ABB RAPID module: Module1.mod

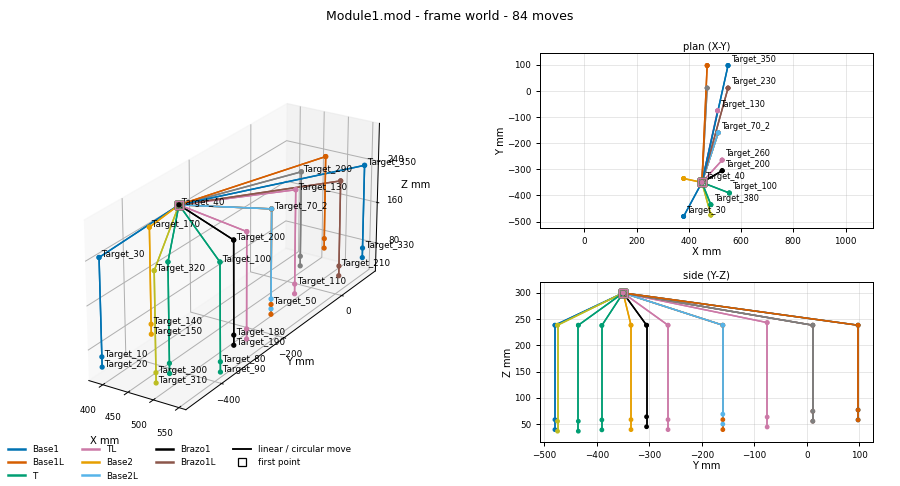
[picture p0: tool path of Module1.mod in frame world, 84 of 86 moves have a stored position in this frame; points joined in program order, loops and branches not executed]
MODULE Module1
        CONST robtarget Target_10:=[[-280,220,28.5],[0,1,0,0],[-1,-2,1,0],[9E+09,9E+09,9E+09,9E+09,9E+09,9E+09]];
    CONST robtarget Target_20:=[[-280,220,9.5],[0,1,0,0],[-1,-2,1,0],[9E+09,9E+09,9E+09,9E+09,9E+09,9E+09]];
    CONST robtarget Target_30:=[[-280,220,208.5],[0,1,0,0],[-1,-1,1,0],[9E+09,9E+09,9E+09,9E+09,9E+09,9E+09]];
    CONST robtarget Target_40:=[[-150,150,270],[0,1,0,0],[-1,-1,1,0],[9E+09,9E+09,9E+09,9E+09,9E+09,9E+09]];
    CONST robtarget Target_50:=[[40,87.5,28.5],[0,1,0,0],[-1,-1,1,0],[9E+09,9E+09,9E+09,9E+09,9E+09,9E+09]];
    CONST robtarget Target_60:=[[40,87.5,9.5],[0,1,0,0],[-1,-1,1,0],[9E+09,9E+09,9E+09,9E+09,9E+09,9E+09]];
    CONST robtarget Target_70:=[[40,87.5,208.5],[0,1,0,0],[-1,-1,1,0],[9E+09,9E+09,9E+09,9E+09,9E+09,9E+09]];
    CONST robtarget Target_80:=[[-190.551,45,28],[0,1,0,0],[0,0,0,0],[9E+09,9E+09,9E+09,9E+09,9E+09,9E+09]];
    CONST robtarget Target_90:=[[-190.551,45,9],[0,1,0,0],[0,0,0,0],[9E+09,9E+09,9E+09,9E+09,9E+09,9E+09]];
    CONST robtarget Target_100:=[[-190.551,45,208],[0,1,0,0],[0,0,0,0],[9E+09,9E+09,9E+09,9E+09,9E+09,9E+09]];
    CONST robtarget Target_110:=[[124.5,90,33.5],[0,-0.707106781,0.707106781,0],[0,0,0,0],[9E+09,9E+09,9E+09,9E+09,9E+09,9E+09]];
    CONST robtarget Target_120:=[[124.5,90,14.5],[0,-0.707106781,0.707106781,0],[0,0,0,0],[9E+09,9E+09,9E+09,9E+09,9E+09,9E+09]];
    CONST robtarget Target_130:=[[124.5,90,213.5],[0,1,0,0],[0,0,0,0],[9E+09,9E+09,9E+09,9E+09,9E+09,9E+09]];
    CONST robtarget Target_140:=[[-135,220,28.5],[0,1,0,0],[-1,-2,1,0],[9E+09,9E+09,9E+09,9E+09,9E+09,9E+09]];
    CONST robtarget Target_150:=[[-135,220,9.5],[0,1,0,0],[-1,-2,1,0],[9E+09,9E+09,9E+09,9E+09,9E+09,9E+09]];
    CONST robtarget Target_160:=[[211.5,50,25.5],[0,0,1,0],[0,0,0,0],[9E+09,9E+09,9E+09,9E+09,9E+09,9E+09]];
    CONST jointtarget JointTarget_3:=[[-34,25,26,0,0,0],[9E+09,9E+09,9E+09,9E+09,9E+09,9E+09]];
    CONST jointtarget JointTarget_4:=[[0,0,0,0,10,0],[9E+09,9E+09,9E+09,9E+09,9E+09,9E+09]];
    CONST robtarget Target_290:=[[211.5,130,208.5],[0,1,0,0],[0,-1,1,0],[9E+09,9E+09,9E+09,9E+09,9E+09,9E+09]];
    CONST robtarget Target_300:=[[-275,115.774,25.5],[0,1,0,0],[0,0,0,0],[9E+09,9E+09,9E+09,9E+09,9E+09,9E+09]];
    CONST jointtarget JointTarget_6:=[[-40.8,22.93,5.77,-27.35,97.75,145],[9E+09,9E+09,9E+09,9E+09,9E+09,9E+09]];
    CONST robtarget Target_70_2:=[[40,87.5,208.5],[0,1,0,0],[-1,-1,1,0],[9E+09,9E+09,9E+09,9E+09,9E+09,9E+09]];
    CONST robtarget Target_170:=[[-135,220,208.5],[0,1,0,0],[0,0,0,0],[9E+09,9E+09,9E+09,9E+09,9E+09,9E+09]];
    CONST robtarget Target_230:=[[211.5,50,208.5],[0,1,0,0],[0,-1,1,0],[9E+09,9E+09,9E+09,9E+09,9E+09,9E+09]];
    CONST robtarget Target_210:=[[211.5,50,44.5],[0,-0.707106781,0.707106781,0],[0,0,2,0],[9E+09,9E+09,9E+09,9E+09,9E+09,9E+09]];
    CONST robtarget Target_220:=[[211.5,50,25.5],[0,-0.707106781,0.707106781,0],[0,0,2,0],[9E+09,9E+09,9E+09,9E+09,9E+09,9E+09]];
    CONST robtarget Target_270:=[[211.5,130,44.5],[0,-0.707106781,0.707106781,0],[0,0,2,0],[9E+09,9E+09,9E+09,9E+09,9E+09,9E+09]];
    CONST robtarget Target_280:=[[211.5,130,25.5],[0,-0.707106781,0.707106781,0],[0,0,2,0],[9E+09,9E+09,9E+09,9E+09,9E+09,9E+09]];
    CONST robtarget Target_320:=[[-275,115.774,208.5],[0,1,0,0],[0,0,0,0],[9E+09,9E+09,9E+09,9E+09,9E+09,9E+09]];
    CONST robtarget Target_310:=[[-275,115.774,6.5],[0,1,0,0],[0,0,0,0],[9E+09,9E+09,9E+09,9E+09,9E+09,9E+09]];
    CONST robtarget Target_350:=[[297.774,50,208.5],[0,1,0,0],[0,-1,1,0],[9E+09,9E+09,9E+09,9E+09,9E+09,9E+09]];
    CONST robtarget Target_330:=[[297.774,50,47],[0,-0.707106781,0.707106781,0],[0,0,2,0],[9E+09,9E+09,9E+09,9E+09,9E+09,9E+09]];
    CONST robtarget Target_340:=[[297.774,50,28],[0,-0.707106781,0.707106781,0],[0,0,2,0],[9E+09,9E+09,9E+09,9E+09,9E+09,9E+09]];
    CONST robtarget Target_410:=[[297.774,130.001,208.5],[0,1,0,0],[0,-1,1,0],[9E+09,9E+09,9E+09,9E+09,9E+09,9E+09]];
    CONST robtarget Target_390:=[[297.774,130.001,47],[0,-0.707106781,0.707106781,0],[0,0,2,0],[9E+09,9E+09,9E+09,9E+09,9E+09,9E+09]];
    CONST robtarget Target_400:=[[297.774,130.001,28],[0,-0.707106781,0.707106781,0],[0,0,2,0],[9E+09,9E+09,9E+09,9E+09,9E+09,9E+09]];
    CONST robtarget Target_380:=[[-235.417,115.774,208.5],[0,1,0,0],[-1,-1,1,0],[9E+09,9E+09,9E+09,9E+09,9E+09,9E+09]];
    CONST robtarget Target_360:=[[-235.417,115.774,25.5],[0,1,0,0],[-1,-1,1,0],[9E+09,9E+09,9E+09,9E+09,9E+09,9E+09]];
    CONST robtarget Target_370:=[[-235.417,115.774,6.5],[0,1,0,0],[-1,-1,1,0],[9E+09,9E+09,9E+09,9E+09,9E+09,9E+09]];
    CONST robtarget Target_430:=[[40,87.5,20],[0,1,0,0],[0,0,0,0],[9E+09,9E+09,9E+09,9E+09,9E+09,9E+09]];
    CONST robtarget Target_440:=[[40,87.5,208.5],[0,1,0,0],[0,0,0,0],[9E+09,9E+09,9E+09,9E+09,9E+09,9E+09]];
    CONST robtarget Target_420:=[[40,87.5,39],[0,1,0,0],[0,0,0,0],[9E+09,9E+09,9E+09,9E+09,9E+09,9E+09]];
    CONST robtarget Target_180:=[[-105.323,72.5,34],[0,1,0,0],[0,0,0,0],[9E+09,9E+09,9E+09,9E+09,9E+09,9E+09]];
    CONST robtarget Target_190:=[[-105.323,72.5,15],[0,1,0,0],[0,0,0,0],[9E+09,9E+09,9E+09,9E+09,9E+09,9E+09]];
    CONST robtarget Target_200:=[[-105.323,72.5,208.5],[0,1,0,0],[0,0,0,0],[9E+09,9E+09,9E+09,9E+09,9E+09,9E+09]];
    CONST robtarget Target_260:=[[-64.44,72.5,208.5],[0,1,0,0],[0,0,0,0],[9E+09,9E+09,9E+09,9E+09,9E+09,9E+09]];
    CONST robtarget Target_240:=[[-64.44,72.5,28.5],[0,1,0,0],[0,0,0,0],[9E+09,9E+09,9E+09,9E+09,9E+09,9E+09]];
    CONST robtarget Target_250:=[[-64.44,72.5,9.5],[0,1,0,0],[0,0,0,0],[9E+09,9E+09,9E+09,9E+09,9E+09,9E+09]];
    CONST jointtarget JointTarget_7:=[[-32,23.81,9.7,-57,45.16,96.13],[9E+09,9E+09,9E+09,9E+09,9E+09,9E+09]];
!***********************************************************
    !
    ! Módulo:  Module1
    !
    ! Descripción:
    !   <Introduzca la descripción aquí>
    !
    ! Autor: Diego
    !
    ! Versión: 1.0
    !
    !***********************************************************


    !***********************************************************
    !
    ! Procedimiento Main
    !
    !   Este es el punto de entrada de su programa
    !
    !***********************************************************
    PROC main()
      SetDO DO_03,0;
        Home;
      WaitDI DI_01,1;
       Acer;
        Base1;
        Base1L;
        T;
        TL;
        Base2;
        Base2L;
        Brazo1;
        Brazo1L;
        Brazo2;
        Brazo2L;
        P1;
        P1L;
        P2;
        P2L;
        Home;
        SetDO DO_03,1;
    ENDPROC
    PROC Base1()
        MoveL Target_40,v150,z100,Hpro\WObj:=Distri2;
        MoveL Target_30,v150,z100,Hpro\WObj:=Distri2;
        MoveL Target_10,v150,z100,Hpro\WObj:=Distri2;
        WaitDI DI_01,1;
       MoveL Target_20,v150,z100,Hpro\WObj:=Distri2;
       WaitTime 1;
        SetDO DO_01,1;
        waittime 0.5;
        SetDO DO_01,0;
        MoveL Target_30,v150,z100,Hpro\WObj:=Distri2;
        MoveL Target_40,v150,z100,Hpro\WObj:=Distri2;
    ENDPROC
    PROC Base1L()
        MoveL Target_40,v150,z100,Hpro\WObj:=Distri2;
        MoveL Target_70_2,v150,z100,Hpro\WObj:=Distri2;
        MoveL Target_50,v150,z100,Hpro\WObj:=Distri2;
        MoveL Target_60,v150,z100,Hpro\WObj:=Distri2;
        WaitTime 1;
        SetDO DO_02,1;
        waittime 0.5;
        SetDO DO_02,0;
        MoveL Target_70,v150,z100,Hpro\WObj:=Distri2;
        MoveL Target_40,v150,z100,Hpro\WObj:=Distri2;
    ENDPROC
    PROC T()
        MoveL Target_40,v150,z100,Hpro\WObj:=Distri2;
        MoveL Target_100,v150,z100,Hpro\WObj:=Distri2;
        MoveL Target_80,v150,z100,Hpro\WObj:=Distri2;
        MoveL Target_90,v150,z100,Hpro\WObj:=Distri2;
        WaitTime 1;
        SetDO DO_01,1;
        waittime 0.5;
        SetDO DO_01,0;
        MoveL Target_100,v150,z100,Hpro\WObj:=Distri2;
        MoveL Target_40,v150,z100,Hpro\WObj:=Distri2;
    ENDPROC
    PROC TL()
        MoveL Target_40,v150,z100,Hpro\WObj:=Distri2;
        MoveL Target_130,v150,z100,Hpro\WObj:=Distri2;
        MoveL Target_110,v150,z100,Hpro\WObj:=Distri2;
        MoveL Target_120,v150,z100,Hpro\WObj:=Distri2;
        WaitTime 1;
        SetDO DO_02,1;
        waittime 0.5;
        SetDO DO_02,0;
        MoveL Target_130,v150,z100,Hpro\WObj:=Distri2;
        MoveL Target_40,v150,z100,Hpro\WObj:=Distri2;
    ENDPROC
    PROC Base2()
        MoveL Target_40,v150,z100,Hpro\WObj:=Distri2;
        MoveL Target_170,v150,z100,Hpro\WObj:=Distri2;
        MoveL Target_140,v150,z100,Hpro\WObj:=Distri2;
        MoveL Target_150,v150,z100,Hpro\WObj:=Distri2;
        WaitTime 1;
        SetDO DO_01,1;
        waittime 0.5;
        SetDO DO_01,0;
        MoveL Target_170,v150,z100,Hpro\WObj:=Distri2;
        MoveL Target_40,v150,z100,Hpro\WObj:=Distri2;
    ENDPROC
    PROC Base2L()
        MoveL Target_40,v150,z100,Hpro\WObj:=Distri2;
        MoveL Target_440,v150,z100,Hpro\WObj:=Distri2;
        MoveL Target_420,v150,z100,Hpro\WObj:=Distri2;
        MoveL Target_430,v150,z100,Hpro\WObj:=Distri2;
        WaitTime 1;
        SetDO DO_02,1;
        waittime 0.5;
        SetDO DO_02,0;
        MoveL Target_440,v150,z100,Hpro\WObj:=Distri2;
        MoveL Target_40,v150,z100,Hpro\WObj:=Distri2;
    ENDPROC
    PROC Brazo1()
        MoveL Target_40,v150,z100,Hpro\WObj:=Distri2;
        MoveL Target_200,v150,z100,Hpro\WObj:=Distri2;
        MoveL Target_180,v150,z100,Hpro\WObj:=Distri2;
        MoveL Target_190,v150,z100,Hpro\WObj:=Distri2;
        WaitTime 1;
        SetDO DO_01,1;
        waittime 0.5;
        SetDO DO_01,0;
        MoveL Target_200,v150,z100,Hpro\WObj:=Distri2;
        MoveL Target_40,v150,z100,Hpro\WObj:=Distri2;
    ENDPROC
    PROC Brazo1L()
        MoveL Target_40,v150,z100,Hpro\WObj:=Distri2;
        MoveL Target_230,v150,z100,Hpro\WObj:=Distri2;
        MoveL Target_210,v150,z100,Hpro\WObj:=Distri2;
        MoveL Target_220,v150,z100,Hpro\WObj:=Distri2;
        WaitTime 1;
        SetDO DO_02,1;
        waittime 0.5;
        SetDO DO_02,0;
        MoveL Target_230,v150,z100,Hpro\WObj:=Distri2;
        MoveL Target_40,v150,z100,Hpro\WObj:=Distri2;
    ENDPROC
    PROC Acer()
        MoveAbsJ JointTarget_7,v1000,z100,Hpro\WObj:=Distri2;
    ENDPROC
    PROC Home()
        MoveAbsJ JointTarget_4,v1000,z100,Hpro\WObj:=Distri2;
    ENDPROC
    PROC Brazo2L()
        MoveL Target_40,v150,z10,Hpro\WObj:=Distri2;
        MoveL Target_290,v150,z0,Hpro\WObj:=Distri2;
        MoveL Target_270,v150,z0,Hpro\WObj:=Distri2;
        MoveL Target_280,v150,z0,Hpro\WObj:=Distri2;
        WaitTime 1;
        SetDO DO_02,1;
        waittime 0.5;
        SetDO DO_02,0;
        MoveL Target_290,v150,z0,Hpro\WObj:=Distri2;
        MoveL Target_40,v150,z0,Hpro\WObj:=Distri2;
    ENDPROC
    PROC P1()
        MoveL Target_40,v150,z10,Hpro\WObj:=Distri2;
        MoveL Target_320,v150,z10,Hpro\WObj:=Distri2;
        MoveL Target_300,v150,z10,Hpro\WObj:=Distri2;
        MoveL Target_310,v150,z10,Hpro\WObj:=Distri2;
        WaitTime 1;
        SetDO DO_01,1;
        waittime 0.5;
        SetDO DO_01,0;
        MoveL Target_320,v150,z10,Hpro\WObj:=Distri2;
        MoveL Target_40,v150,z10,Hpro\WObj:=Distri2;
    ENDPROC
    PROC P1L()
        MoveL Target_40,v150,z10,Hpro\WObj:=Distri2;
        MoveL Target_350,v150,z10,Hpro\WObj:=Distri2;
        MoveL Target_330,v150,z10,Hpro\WObj:=Distri2;
        MoveL Target_340,v150,z10,Hpro\WObj:=Distri2;
        WaitTime 1;
        SetDO DO_02,1;
        waittime 0.5;
        SetDO DO_02,0;
        MoveL Target_350,v150,z10,Hpro\WObj:=Distri2;
        MoveL Target_40,v150,z10,Hpro\WObj:=Distri2;
    ENDPROC
    PROC P2L()
        MoveL Target_40,v150,z10,Hpro\WObj:=Distri2;
        MoveL Target_410,v150,z10,Hpro\WObj:=Distri2;
        MoveL Target_390,v150,z10,Hpro\WObj:=Distri2;
        MoveL Target_400,v150,z10,Hpro\WObj:=Distri2;
        WaitTime 1;
        SetDO DO_02,1;
        waittime 0.5;
        SetDO DO_02,0;
        MoveL Target_410,v150,z10,Hpro\WObj:=Distri2;
        MoveL Target_40,v150,z10,Hpro\WObj:=Distri2;
    ENDPROC
    PROC P2()
        MoveL Target_40,v150,z10,Hpro\WObj:=Distri2;
        MoveL Target_380,v150,z10,Hpro\WObj:=Distri2;
        MoveL Target_360,v150,z10,Hpro\WObj:=Distri2;
        MoveL Target_370,v150,z10,Hpro\WObj:=Distri2;
        WaitTime 1;
        SetDO DO_01,1;
        waittime 0.5;
        SetDO DO_01,0;
        MoveL Target_380,v150,z10,Hpro\WObj:=Distri2;
        MoveL Target_40,v150,z10,Hpro\WObj:=Distri2;
    ENDPROC
    LOCAL PROC Brazo2()
        MoveL Target_40,v150,z0,Hpro\WObj:=Distri2;
        MoveL Target_260,v150,z0,Hpro\WObj:=Distri2;
        MoveL Target_240,v150,z0,Hpro\WObj:=Distri2;
        MoveL Target_250,v150,z0,Hpro\WObj:=Distri2;
        WaitTime 1;
        SetDO DO_01,1;
        waittime 0.5;
        SetDO DO_01,0;
        MoveL Target_260,v150,z0,Hpro\WObj:=Distri2;
        MoveL Target_40,v150,z0,Hpro\WObj:=Distri2;
    ENDPROC
ENDMODULE
